// TIA Portal V20 export
DATA_BLOCK "dHMI"   // DB30151
{ S7_Optimized_Access := 'TRUE' }
// stored: AutoNumber false, MemoryReserve 100
   VAR
      HMI_SCREEN_Change : Array[1..4] of Int;
      HMI_SCREEN_NUM : Array[1..5] of Int;
   END_VAR
BEGIN
END_DATA_BLOCK
